{attribute 'GeneratedUsingTerminal: BK1250-0000-0019'}
{attribute addProperty BoxType "BK1250-0000-0019"}
{attribute addProperty Id "Term_388_KL1002KL1002_BB38DA8F0"}
{attribute addProperty CRC "3709641895"}
{attribute addProperty Size "0"}
TYPE A_0018_BK1250_0000_0019_DD1CA4A7 EXTENDS BK1250_A2FCADE7 :
STRUCT
	{attribute addProperty Name "Term_388_KL1002"}
	Term_388_KL1002 : KL1002_BB38DA8F;
END_STRUCT
END_TYPE

(* stored: Version 1.2.0.0, ProductVersion 3.1.4024.9
   DUT A_0018_BK1250_0000_0019_DD1CA4A7: Id {0cd0df37-430a-4d83-9742-7e1f6f37d0da} *)
